Europa
• Zürich, Schweiz: Eidgenössischen Technischen Hochschule Zürich
129.132.98.11: bernina.ethz.ch
Servicebereich: Schweiz und Europa  
• Standort: Kopenhagen, Dänemark, Europa 
clock.netcetera.dk; clock2.netcetera.dk 
Servicebereich: Dänemark, Skandinavien und Nordeuropa  
• Spanien: Altea 
slug.ctv.es
Servicebereich: Spanien  
• Pieksamaki, Finnland: Keski-Savon Oppimiskeskus
tick.keso.fi; tock.keso.fi
Servicebereich: Finnland  
• Meudon, Frankreich: Observatoire de Paris-Meudon 
ntp.obspm.fr 
Servicebereich: Frankreich und Europa  
• Lyon, Frankreich: CISM 
ntp.univ-lyon1.fr 
Servicebereich: Frankreich, Schweiz, Italien und Europa  
• Paris, Frankreich: VIA, Ecole Centrale
138.195.130.70: ntp.via.ecp.fr
Servicebereich: Frankreich und Europa  
• Budapest, Ungarn: KFKI Research Institute for Particle and Nuclear Physics
148.6.0.1: time.kfki.hu
Servicebereich: HUNGARNET  
• Italien: Net4u Srl, Vercelli, Italien
195.32.52.129: ntps.net4u.it
Servicebereich: Italien  
• Oslo, Norwegen: Universität Oslo
129.240.64.3: fartein.ifi.uio.no 
Servicebereich: NORDUnet  
• Oslo, Norwegen: Alcanet International
time.alcanet.no
Servicebereich: Europa 
• Krakau, Polen: Academic Computer Centre 
149.156.4.11: info.cyf-kr.edu.pl
Servicebereich: Polen und Europa  
• Lund, Schweden: Lund Institute of Technology
130.235.20.3: ntp.lth.se 
Servicebereich: Schweden und NORDUnet 
• Ljubljana, Slowenien: Institute of Biophysics, University of Ljubljana
biofiz.mf.uni-lj.si 193.2.69.11
Servicebereich: Slowenien und Europa  
• Ljubljana, Slowenien: Hydrometeorological Institute of Slovenia
hmljhp.rzs-hm.si
Servicebereich: Slowenien und Europa  
• Ljubljana, Slowenien: Academic and Research Network of Slovenia
ntp1.arnes.si; ntp2.arnes.si
Servicebereich: Slowenien und Europa  
• Ljubljana, Slowenien: J. Stefan Institute
time.ijs.si
Servicebereich: Slowenien und Europa  

Britische Inseln
• Dublin, Irland: School of Mathematics, Trinity College 
ntp.cs.tcd.ie; ntp.maths.tcd.ie; ntp.tcd.ie
Servicebereich: Irland und Großbritannien 
• Glasgow, Schottland: Strathclyde University 
ntp.cs.strath.ac.uk 
Servicebereich: Großbritannien, Europa und andere 
• Cambridge, Großbritannien
ntp0.uk.uu.net; ntp1.uk.uu.net; 
ntp2.uk.uu.net 
Servicebereich: UUNET (in Großbritannien früher auch als PIPEX bekannt) und Großbritannien.  
• Manchester, England: University of Manchester
ntp2a.mcc.ac.uk; ntp2b.mcc.ac.uk;
ntp2c.mcc.ac.uk; ntp2d.mcc.ac.uk 
Servicebereich: Großbritannien  
• Buckinghamshire, Großbritannien: Wibble U.K., Aylesbury
tick.tanac.net
Servicebereich: Großbritannien  

Asien
• Moskau, Russland: Landau Institute for Theoretical Physics
193.233.9.7: ntp.landau.ac.ru
Servicebereich: Russland  
• Russland: Pushchino (bei Moskau)
194.149.67.130: ntp.psn.ru
Servicebereich: Russland 
• Chernogolovka, Russland: Chernogolovka Scientific Center (bei Moskau)
193.233.46.10: sign.chg.ru
Servicebereich: Russland  

Fernost und pazifische Randgebiete
• Tokyo, Japan: Cyber Fleet, Inc.
203.139.30.195: ntp.cyber-fleet.net
Servicebereich: Japan und Ostasien  
• Seoul, Korea: Inet, Inc.
time.nuri.net
Servicebereich: Korea, Japan, Hong Kong und Ostasien  
• Hamilton, Neuseeland: Universität Waikato
truechimer.waikato.ac.nz; truechimer1.waikato.ac.nz; 
truechimer2.waikato.ac.nz; truechimer3.waikato.ac.nz
Servicebereich: Neuseeland  
• Singapur und Philippinen: 
ntp.shim.org 
Servicebereich: Singapur  

Afrika
• Lagos, Nigeria: Supernet300
ntp.supernet300.com
Servicebereich: Westafrika (hauptsächlich nigerischer NITEL-Backbone)  
• Pietermaritzburg, Südafrika: Natal University
143.128.82.200: ntp.cs.unp.ac.za
Servicebereich: Südafrika  

Australien
• Adelaide, Südaustralien: University of Adelaide
129.127.28.4: augean.eleceng.adelaide.edu.au
129.127.40.3: ntp.adelaide.edu.au
203.21.37.18: ntp.saard.net
Servicebereich: AARNet  
• Carlton, Victoria, Australien: eSec Limited
203.21.84.4: time.esec.com.au  

*)

*)
END_FUNCTION_BLOCK

(* POU Logic/gate logic/Swap_Byte, ST *)
FUNCTION Swap_Byte : WORD
VAR_INPUT
	IN : WORD;
END_VAR
VAR
END_VAR

(*
version 1.0	4 feb 2008
programmer 	hugo
tested by		tobias

This function swaps the high and low byte of the word in.

*)
Swap_Byte := ROL(in,8);


(* revision history
hm		4. feb 2008	rev 1.0
	original version

*)
END_FUNCTION

(* POU Logic/gate logic/Swap_Byte2, ST *)
FUNCTION Swap_Byte2 : DWORD
VAR_INPUT
	IN : DWORD;
END_VAR
VAR
END_VAR

(*
version 1.0	4 feb 2008
programmer 	hugo
tested by		tobias

This function reverses the byte order in the dword.

*)
Swap_Byte2 := (ROR(in,8) AND 16#FF00FF00) OR (ROL(in,8) AND 16#00FF00FF);

(* revision history
hm		4. feb 2008	rev 1.0
	original version

*)
END_FUNCTION

(* POU Logic/generators/TONOF, ST *)
FUNCTION_BLOCK TONOF
VAR_INPUT
	IN : BOOL;
	T1, T2 : TIME;
END_VAR
VAR_OUTPUT
	Q : BOOL;
END_VAR
VAR
	X : TON;
	Y : TOF;
END_VAR

(*
version 1.1	17 sep 2007
programmer 	hugo
tested by		tobias

TONOF generated a TON and TOF Delay for the Input N TON (T1) and TOF (T2) can be configured separately
*)
X(IN := IN, PT := T1);
Y(in := X.Q, PT := T2);
Q := Y.Q;

(* revision history
hm	10. dec 2007	rev 1.0
	original version

*)
	
END_FUNCTION_BLOCK

(* POU String/trim1, ST *)
FUNCTION trim1 : STRING
VAR_INPUT
	str : STRING;
END_VAR
VAR
	pos: INT;
END_VAR

(*
version 1.0	4 feb 2008
programmer 	hugo
tested by		tobias

the function replaces all multiple blanks within a string by only one blank.
leading and ending blanks will be deleted

*)
trim1 := str;
REPEAT
	pos := FIND(trim1,'  ');
	trim1 := REPLACE(trim1,' ',2,pos);
UNTIL pos = 0	END_REPEAT;
(* beginning and ending blanks need to be stripped off *)
IF LEFT(trim1,1) = ' ' THEN trim1 := DELETE(trim1,1,1); END_IF;
IF RIGHT(trim1,1) = ' ' THEN trim1 := DELETE(trim1,1,LEN(trim1)); END_IF;


(* revision histroy
hm		4. feb. 2008		rev 1.0
	original release

*)	
END_FUNCTION

(* POU engineering/signal processing/Word_to_Range, ST *)
FUNCTION Word_to_Range : REAL
VAR_INPUT
	X : WORD;
	low : REAL;
	high : REAL;
END_VAR
VAR
END_VAR

(*
version 1.0	9. jan 2008
programmer 	hugo
tested by		tobias

Word_to_Range converts a Byte into a real between low and high.

*)
Word_to_Range := (high - low) * X / 65535.0 + low;


(* revision history
hm	9. jan 2008		rev 1.0
	original version

*)
END_FUNCTION

(* POU XTEST/Baustein Tests/work_week_test, ST *)
FUNCTION_BLOCK work_week_test
VAR_INPUT
END_VAR
VAR_OUTPUT
	error : BOOL;
	dx: DATE;
END_VAR
VAR
	y : ARRAY[0..30] OF INT := 1990,1991,1992,1993,1993,1994,1994,1995,1995,1996,1997,1998,1999,1999,2000,2000,2001,2002,2003,2004,2005,2005,2006,2006,2007,2008,2009,2010,2010,2011,2011;
	w : ARRAY[0..30] OF INT := 1,	1,	 1,   53,  1,   52,	 1,   52,  1,   1,   1,   1,   53,  1,   52,  1,   1,   1,   1,   1,   53,  1,   52,  1,   1,	1,   1,	  53,  1,   52,  1;
	d : ARRAY[0..30] OF INT := 7,	6,	 5,	  3,   10,  2,   9,   1,   8,   7,   5,   4,   3,   10,  2,   9,   7,   6,   5,   4,   2,   9,   1,   8,   7,	6,	 4,	  3,   10,  2,   9;
	i: INT;
	comp: INT;
	d1: DATE;
	day: INT;
	week: INT;
	yr: INT;
END_VAR
IF error THEN RETURN; END_IF;

FOR i := 0 TO 30 DO
	day := d[i];
	week := w[i];
	yr := y[i];
	d1 := set_Date(yr,1,day);
	comp := work_week(d1);
	IF comp <> week THEN
		error := TRUE;
		dx := d1;
	END_IF;
	d1 := date_add(d1,-6,0,0,0);
	comp := work_week(d1);
	IF comp <> week THEN
		error := TRUE;
		dx := d1;
	END_IF;

END_FOR;
END_FUNCTION_BLOCK

(* POU XTEST/Baustein Tests/year_test, ST *)
FUNCTION year_test : BOOL
VAR_INPUT
END_VAR
VAR
	x : BOOL := TRUE;
	i: INT;
	jan1: DATE;
	dez31: DATE;
END_VAR
FOR i := 1980 TO 2099 DO
	jan1 := set_Date(i,1,1);
	dez31 := set_Date(i,12,31);
	x := X AND year(jan1) = i AND year(dez31) = i;
END_FOR;
year_test := x;
END_FUNCTION
